PROGRAM MAIN

VAR

bButton_1 	: BOOL	:=	FALSE; // INOUT SIGNAL FROM BUTTON 1 
bLamp_1 		: BOOL	:=	FALSE; // OUTPUT SIGNAL

END_VAR

bLamp_1 := bButton_1;

END_PROGRAM

(* stored: Version 1.1.0.1, ProductVersion 3.1.4026.18
   POU MAIN: Id {30233d5b-b8c4-41d3-a608-5078909698a6}, SpecialFunc None *)
